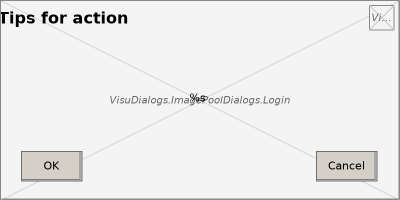
VISUALIZATION WARM  // 400x200
VAR_IN_OUT
	warmHMI:WARMStruct;
END_VAR
    Image (0,0 400x200), image: VisuDialogs.ImagePoolDialogs.Login
    Button (21,151 61x30), "OK"
        OnMouseClick: execute { warmHMI.bOK:=TRUE; warmHMI.showFlag:=FALSE; }
    Button (316,151 61x30), "Cancel"
        OnMouseClick: execute { warmHMI.bNO:=TRUE; warmHMI.showFlag:=FALSE; }
    Rectangle (24,83 347x30), "%s", text variable: warmHMI.showText
    Image (369,5 25x25), image: VisuDialogs.ImagePoolDialogs.Delete
        OnMouseClick: execute { warmHMI.bNO:=TRUE; warmHMI.showFlag:=FALSE; }
    Label (5,3 116x30), "Tips for action"
END_VISUALIZATION

(* stored: Version 1.1.0.1, ProductVersion 3.1.4024.4
   Visu WARM: Id {dcc6b9f5-f672-4180-91f9-a591f80647aa} *)
